Staubli VAL3: editNum.pgx

public program editNum(string& x_sItem (dimensions=1), string& x_sItemValue (dimensions=1), num& x_nValue (dimensions=1), num x_nSelect (dimensions=1), num x_nMin (dimensions=1), num x_nMax (dimensions=1))
  local string l_sEmpty
  local num l_nValue
  local bool l_bRes
  local num l_nKey
  local num l_nPos
begin
  //
  do
    //    call clear(0,13)
    call findPos(x_sItem,":",l_nPos)
    gotoxy(nTopX+1,nTopY+nView+1)
    setTextMode(0)
    put(x_sItem)
    call strlength(l_sEmpty,nBottomX-l_nPos+1)
    call type(nTopX+l_nPos+2,nTopY+nView+1,l_sEmpty)
    gotoxy(nTopX+l_nPos+2,nTopY+nView+1)
    toNum(x_sItemValue,l_nValue,l_bRes)
    l_nKey=get(l_nValue)
    if l_nKey==270
      if x_nMin<x_nMax
        if l_nValue<x_nMin or l_nValue>x_nMax
          popUpMsg("取值范围:"+toString(".1",x_nMin)+"到"+toString(".1",x_nMax))
        else
          x_sItemValue=toString(".3",l_nValue)
          x_nValue=l_nValue
        endIf
      else
        x_sItemValue=toString(".3",l_nValue)
        x_nValue=l_nValue
      endIf
    endIf
    call strfill(x_sItem,l_nPos+1,x_sItem)
    x_sItem=x_sItem+x_sItemValue
    call strlength(x_sItem,nBottomX+1)
    gotoxy(nTopX+1,nTopY+nView+1)
    setTextMode(1)
    call type(nTopX+1,nTopY+nView+1,x_sItem)
    setTextMode(0)
    delay(0)
  until l_nKey==270 or l_nKey==255
end
